TYPE ST_AxisConfig :
STRUCT
    (* Soft limits *)
    minPosition: REAL;
    maxPosition: REAL;

    (* Motion parameters *)
    targetPosition: REAL;
    targetVelocity: REAL := 0.2;
    jogStep: REAL;

    (* SetPosition *)
    positionSetValue: REAL;

    (* LVDT sensor *)
    lvdtThreshold: REAL;
    lvdtFunctionOn: BOOL := TRUE;
    lvdtManualReleaseAlarm: BOOL;
    scalingFactor_LVDT: REAL := 1;

    (* Position retain (survives power cycle) *)
    currentPositionRetain: REAL;

    (* Axis name for error messages *)
    name: STRING(30);
	
	(* backlash *)
	backlash: REAL:=0.2;          (* mm, 默认 0 *)
	backlashEnable: BOOL;    (* 默认 FALSE *)

END_STRUCT
END_TYPE

(* stored: Version 1.1.0.1, ProductVersion 3.1.4024.6
   DUT ST_AxisConfig: Id {5e7afc7f-fbae-421a-9118-4f359d353de0} *)
